TYPE Objet_Mot_TOR :
STRUCT
		Mot_Lecture 	:INT; (*Mot de lecture des bits*)
		Mot_Ecriture 	:INT; (*Mot d'écriture des bits*)
END_STRUCT
END_TYPE

(* stored: Version 1.1.0.1, ProductVersion 3.1.4024.12
   DUT Objet_Mot_TOR: Id {f028d1ad-a15c-4e4b-963a-da87bca5a77e} *)
